% RSLogix 500 project Job XX - Alternating Forward Reverse.RSS, saved by version 10.00.00.00 %
PROJECT "UNTITLED"    % processor: Bul.1763 MicroLogix 1100 Series B %

PROGRAM FILES
  LAD 2   4 rungs

DATA FILES
  O0 OUTPUT  4 elements
  I1 INPUT  6 elements
  S2 STATUS  66 elements
  B3 BINARY  1 elements
  T4 TIMER  1 elements
  C5 COUNTER  1 elements
  R6 CONTROL  1 elements
  N7 INTEGER  1 elements
  F8 FLOAT  1 elements

LADDER 2
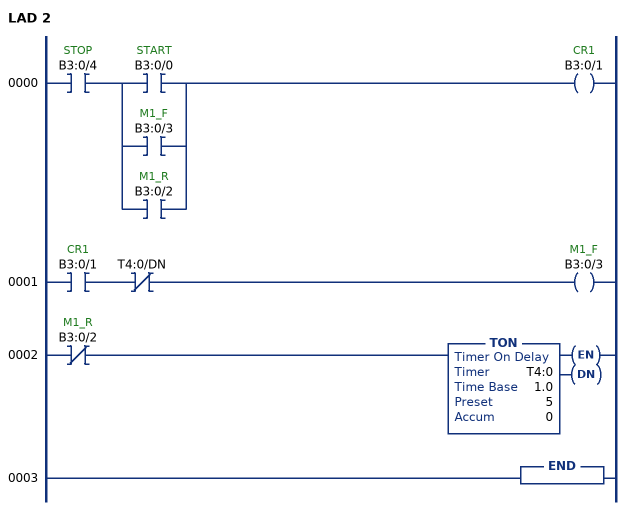
% Rung: 0 %  % edit flag set %
SOR XIC B3:0/4 BST XIC B3:0/0 NXB XIC B3:0/3 NXB XIC B3:0/2 BND OTE B3:0/1 EOR
%   B3:0/4  STOP %
%   B3:0/0  START %
%   B3:0/3  M1_F %
%   B3:0/2  M1_R %
%   B3:0/1  CR1 %
% Rung: 1 %
SOR XIC B3:0/1 XIO T4:0/DN OTE B3:0/3 EOR
%   B3:0/1  CR1 %
%   B3:0/3  M1_F %
% Rung: 2 %
SOR XIO B3:0/2 TON T4:0 1.0 5 0 EOR
%   B3:0/2  M1_R %
% Rung: 3 %
SOR END EOR

DATA TABLE (non-zero values as saved)
DATA T4
% .PRE .ACC %
% T4:0 % 5 0
